{attribute 'qualified_only'}
VAR_GLOBAL
	bSystemStart : BOOL := FALSE; 			//HMI Start
    bAutoMode : BOOL := FALSE;				//HMI Auto
    bCNCOn : BOOL := FALSE;					//HMI CNC ON
    bRetrieveCMD : BOOL := FALSE;			//HMI Retrieve command
    bReset : BOOL := FALSE;					//HMI Reset

    iProductID : INT := 4000;				//Current Product ID
    arrStoredIDs : ARRAY[1..15] OF INT := [0];		//Array of stored products
    arrExitIDs : ARRAY[1..15] OF INT:= [0];		//Array of exited products
    iStorageCount : INT := 0;				//num of stored items
    iExitCount : INT := 0;					//num of retrieved items

    bFaultDetected : BOOL := FALSE;			//global fault indicator
    sFaultMessage : STRING := '';			//global fault message
	
	// Indicates System is in run state
	SystemRun: BOOL := FALSE;
	// Box ID of queued Container
	QueuedBoxID: INT := 0;
	// Box Waiting for crane
	ContainerWaitingInput: BOOL := FALSE;
	
	ContainerWaitingOutput : BOOL := FALSE;
	
	//Warehouse has reached 15 box capacity
	WarehouseFull : BOOL := FALSE;
	
	//If crane is in input mode
	InputtingBoxes : BOOL := TRUE;
	//If crane is in output mode
	OutputtingBoxes : BOOL := FALSE;
	//Commanded location of crane
	CommandedLocation : INT :=1;
END_VAR

(* stored: Version 1.1.0.1
   GVL GVL: Id {0c821d1f-093b-4240-bec7-e300c6a1078a} *)
